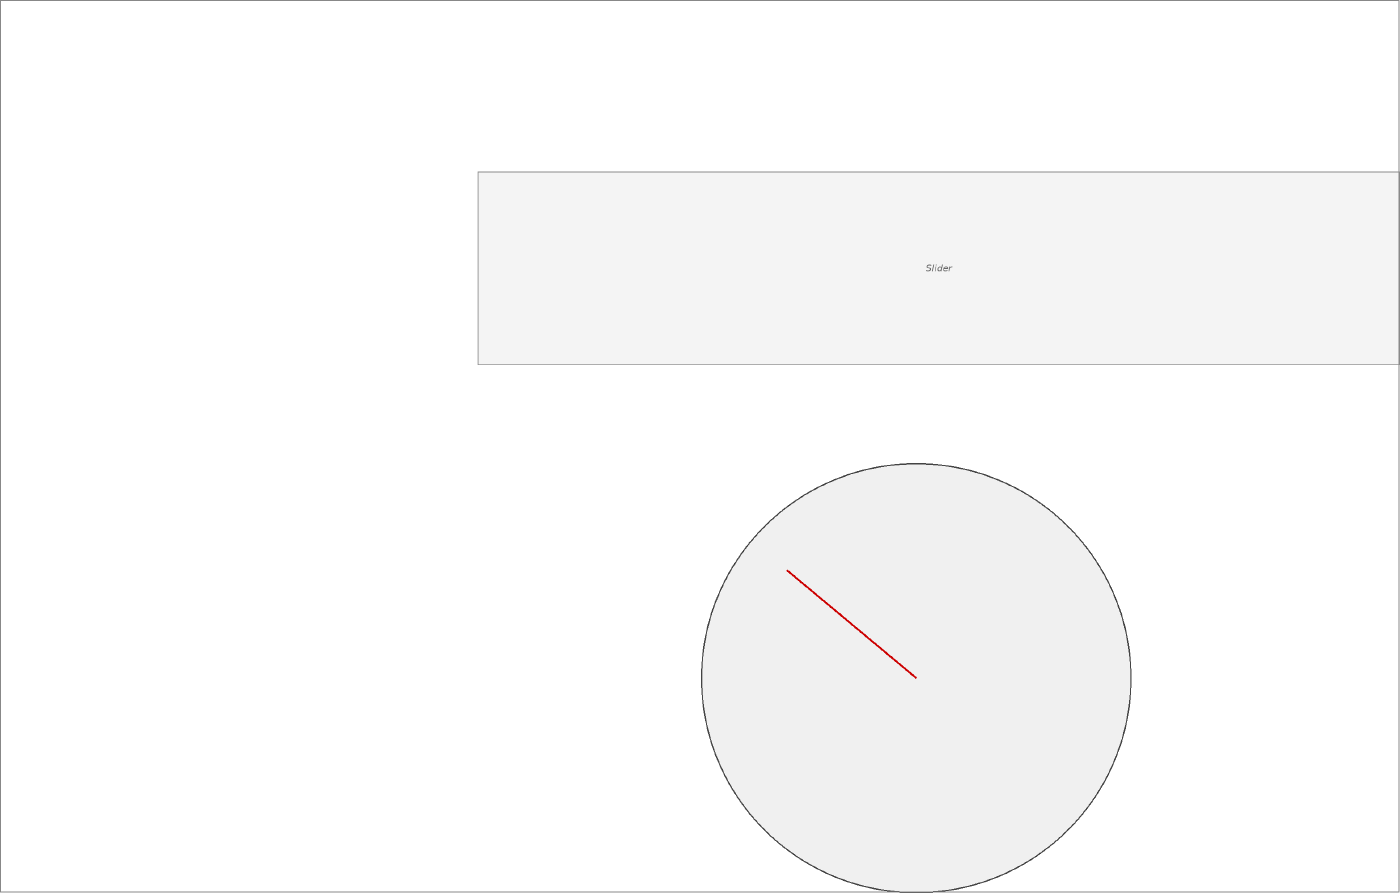
VISUALIZATION Visualization  // 1565x999
    Slider (534,192 1031x216), variable: MAIN.intUltrasonicSensor, scale 0..100
        p2541109501: MAIN.voltageUltrasonicSensor
    Meter180 (586,518 876x481), value: MAIN.voltageUltrasonicSensor, style: Meter-Meter180-Gray, scale format: %.1f, scale 0..10
END_VISUALIZATION

(* stored: Version 1.1.0.1, ProductVersion 3.1.4024.13
   Visu Visualization: Id {35940344-55f9-4bfa-bf63-02b397c6610f} *)
